(* CoDeSys 2.3.9.42 project: CR0403 AGV.pro *)
(* Libraries: SysLibPlcCtrl.lib 13.6.03 15:49:00, SysLibFile.lib 23.9.04 10:11:36, SysLibTime.lib 27.4.05 10:36:52, SysLibTargetVisu.lib 5.4.04 13:31:00, LinuxSystemLib.Lib 18.3.03 13:26:50, ifm_pdm_file_V010006.lib 14.1.08 14:21:32, ifm_CR0403\ifm_CR0403_V030100.lib 22.3.17 12:39:40, Util.lib 6.11.07 16:39:24, ifm_J1939_NT\ifm_J1939_NT_V020004.lib 18.9.14 16:13:02, ifm_RAWCan\ifm_RAWCan_NT_V020004.lib 3.11.15 19:07:52, standard.lib 4.10.05 11:14:46, SysLibCallback.lib 26.9.08 17:43:52 *)

(* PLC configuration (modules and I/O channels)
Configuration [LocalConfiguration] node 0, in %IB0 out %QB0 {IFM_PARAM_WORD_TIME = 0}
Input/Output [LocalInputOutput] node 1, in %IB0 out %QB0
  Inputs Binary [LocalIn] node 0, in %IB0 out %QB0
    IN00 AT %IB0 [ChInputBool] Input 00 Bit
    IN01 AT %IB1 [ChInputBool] Input 01 Bit
    IN02 AT %IB2 [ChInputBool] Input 02 Bit
    IN03 AT %IB3 [ChInputBool] Input 03 Bit
    IN04 AT %IB4 [ChInputBool] Input 04 Bit
    IN05 AT %IB5 [ChInputBool] Input 05 Bit
    IN06 AT %IB6 [ChInputBool] Input 06 Bit
    IN07 AT %IB7 [ChInputBool] Input 07 Bit
    IN08 AT %IB8 [ChInputBool] Input 08 Bit
    IN09 AT %IB9 [ChInputBool] Input 09 Bit
    IN10 AT %IB10 [ChInputBool] Input 10 Bit
    IN11 AT %IB11 [ChInputBool] Input 11 Bit
  Outputs Binary [LocalOut] node 1, in %IB12 out %QB0
    OUT00 AT %QB0 [ChOutputBool] Output 00 Bit
    OUT01 AT %QB1 [ChOutputBool] Output 01 Bit
    OUT02 AT %QB2 [ChOutputBool] Output 02 Bit
    OUT03 AT %QB3 [ChOutputBool] Output 03 Bit
    OUT04 AT %QB4 [ChOutputBool] Output 04 Bit
    OUT05 AT %QB5 [ChOutputBool] Output 05 Bit
    OUT06 AT %QB6 [ChOutputBool] Output 06 Bit
    OUT07 AT %QB7 [ChOutputBool] Output 07 Bit
    OUT08 AT %QB8 [ChOutputBool] Output 08 Bit
    OUT09 AT %QB9 [ChOutputBool] Output 09 Bit
    OUT10 AT %QB10 [ChOutputBool] Output 10 Bit
    OUT11 AT %QB11 [ChOutputBool] Output 11 Bit
  System Inputs [LocalSystemInputs] node 2, in %IB12 out %QB12
    SUPPLY_VOLTAGE_VBBS AT %IW6 [ChInputWord] Supply voltage VBBS
    SUPPLY_VOLTAGE_VU AT %IW7 [ChInputWord] Supply voltage VU
    SUPPLY_VOLTAGE_VBB1 AT %IW8 [ChInputWord] Supply voltage VBB1
    SUPPLY_VOLTAGE_VBB2 AT %IW9 [ChInputWord] Supply voltage VBB2
    TEMPERATURE AT %IW10 [ChInputInt] Temperature
J1939 Interface [CAN_J1939] node 1, in %IB32 out %QB12
CANopen Interface [CAN_OPEN] node 0, in %IB32 out %QB12
J1939 Interface [CAN_J1939] node 1, in %IB32 out %QB12
*)

(* Global variable list: Global_Variables *)
VAR_GLOBAL
	Route1: ARRAY [1..2,1..4] OF REAL := 10, 100, 100, 10, 10, 10, 100, 100;
END_VAR

(* Data type *)
TYPE CONSTANTS_MATH :
STRUCT
	RadDeg : REAL := 57.29577951; (*Conversie van radialen naar degrees*)
	PI : REAL := 	3.14159265358979323846264338327950288;		(* Kreiszahl PI *)
	PI2 : REAL := 	6.28318530717958647692528676655900576;	(* PI * 2 *)
	PI4 : REAL :=  12.56637061435917295385057353311801152;	(* PI * 4 *)
	PI05 : REAL :=  1.5707963267949;							(* PI / 2 *)
	PI025 : REAL := 0.785398163397448;							(* PI / 4 *)
	PI_INV : REAL := 0.318309886183791;						(* 1 / PI *)
	E : REAL := 	2.71828182845904523536028747135266249;		(* Euler constant e *)
	E_INV : REAL := 0.367879441171442;							(* 1 / e *)
	SQ2 : REAL :=	1.4142135623731;							(* Wurzel von 2 *)
	FACTS : ARRAY[0..12] OF DINT := 1,1,2,6,24,120,720,5040,40320,362880,3628800,39916800,479001600;
END_STRUCT
END_TYPE

(* POU PLC_PRG, ST *)
PROGRAM PLC_PRG
VAR
	CAN_ENABLE_CAN2: CAN_ENABLE;
	CAN_ENABLE_CAN1: CAN_ENABLE;

END_VAR
CAN_ENABLE_CAN1(ENABLE:=TRUE , CHANNEL:=1 , BAUDRATE:=500 , RESULT=> );

CAN_RX_comm_display();

NavSof();

PosEncoderLinks;


PosEncoderRechts;
END_PROGRAM

(* POU CAN_RX_comm_display, ST *)
PROGRAM CAN_RX_comm_display
VAR
	CAN_RX_comm_keys_display: CAN_RX;
	UNPACK_comm_keys: UNPACK;
	keyF1: BOOL;
	keyF2: BOOL;
	keyF3: BOOL;
	keyF4: BOOL;
END_VAR
CAN_RX_comm_keys_display(
	ENABLE:=TRUE ,
	CHANNEL:=1 ,
	ID:=16#190 ,
	DATA=> ,
	RESULT=> );

IF CAN_RX_comm_keys_display.RESULT=1  THEN

UNPACK_comm_keys(
	B:=CAN_RX_comm_keys_display.DATA[0] ,
	B0=>keyF1 ,
	B1=>keyF2 ,
	B2=>keyF3,
	B3=>keyF4 ,
	B4=> ,
	B5=> , 
	B6=> , 
	B7=> );


END_IF

IF keyF1 THEN
OUT00:=TRUE;
ELSE
OUT00:=FALSE;
END_IF

IF keyF2 THEN
OUT01:=TRUE;
ELSE
OUT01:=FALSE;
END_IF
END_PROGRAM

(* POU NavSof, ST *)
PROGRAM NavSof
VAR
	(*Variabelen voor het binnen lezen van de UWB data via de CAN bus*)
	CAN_RX_POZXY_COORD: CAN_RX;							(*FB om een CAN bericht binnen te lezen*)
	ARRAY_TO_DWORD_Xcoor: ARRAY_TO_DWORD;				(*Data van een ARRAY naar een getal omvormen*)
	xHuidigeCoordinaat: REAL;										(*Datatype vastleggen*)
	ARRAY_TO_DWORD_Ycoor: ARRAY_TO_DWORD;
	yHuidigeCoordinaat: REAL;

	(*Variabelen NavSof*)
	i_Waypoints: INT := 0;													(*Variabele die het aantal waypoints van onze huidige route bevat*)
	x_Jumplock: BOOL := TRUE;											(*Flag zodat bij opstart éénmalig X en Y-huidig kunnen gebruikt worden als X en Y start voor de trackline*)
	xStartCoordinaat: REAL := 0;											(*X coordinaat voor begin trackline*)
	yStartCoordinaat: REAL := 0;											(*Y coordinaat voor einde trackline*)
	xEindCoordinaat: REAL := 0;											(*X coordinaat voor einde trackline*)
	yEindCoordinaat: REAL := 0;											(*Y coordinaat voor einde trackline*)
	rAfstandTotWaypoint: REAL := 0;										(*Bevat de afstand tot het waypoint*)
	rTrackHoek: REAL:= 0;												(*Bevat de trackhoek, de hoek die de AGV naar links of rechts doet sturen opdat deze terug op de trackline zou uitkomen*)
	CONSTANTS_MATH: CONSTANTS_MATH;							(*Struct die bepaalde wiskundige constanten bevat*)


	rHoekAGV: REAL;
	rTrack: REAL;
	BNO_lock: BOOL;
	StuurLinks: REAL;
	beginBNO: REAL;
	eindeBNO: REAL;
	StuurNeutraal: REAL;
END_VAR
(*Binnenlezen van de huidige positie d.m.v. UWB*)
CAN_RX_POZXY_COORD(
	ENABLE:= TRUE,
	CHANNEL:=1 ,
	ID:=16#A1 ,
	DATA=> , 
	RESULT=> );

IF  CAN_RX_POZXY_COORD.RESULT=1 THEN

ARRAY_TO_DWORD_Xcoor(
	Byte_0:=CAN_RX_POZXY_COORD.DATA[0] ,
	Byte_1:=CAN_RX_POZXY_COORD.DATA[1] ,
	Byte_2:=CAN_RX_POZXY_COORD.DATA[2] ,
	Byte_3:=CAN_RX_POZXY_COORD.DATA[3] ,
	DWORD_OUT=> xHuidigeCoordinaat );

ARRAY_TO_DWORD_Ycoor(
	Byte_0:=CAN_RX_POZXY_COORD.DATA[4] ,
	Byte_1:=CAN_RX_POZXY_COORD.DATA[5] ,
	Byte_2:=CAN_RX_POZXY_COORD.DATA[6] ,
	Byte_3:=CAN_RX_POZXY_COORD.DATA[7] ,
	DWORD_OUT=> yHuidigeCoordinaat );

END_IF

(*Het aantal waypoints van onze huidige route bepalen*)
i_Waypoints := SIZEOF(Route1)/8;							(*Route 1 bevat 2 * 4 coordinaten die telkens 4 bytes (datatype REAL) innemen
																de totale grootte van deze array is dus 32 bytes / 8 geeft ons het aantal waypoints*)

(*Ervoor zorgen dat bij opstart éénmalig X- en Y-huidig gebruikt kunnen worden als X- en Y-start voor de trackline*)
IF x_Jumplock = TRUE
THEN
	xStartCoordinaat := xHuidigeCoordinaat;
	yStartCoordinaat := yHuidigeCoordinaat;
	x_Jumplock := FALSE;
END_IF;

(*Uitrekenen wat de afstand tot het volgende waypoint is*)
rAfstandTotWaypoint := Afstand_Punt_Punt(xStartCoordinaat, yStartCoordinaat, xEindCoordinaat, yEindCoordinaat);

(*Ervoor zorgen dat bij het afleggen van een route er steeds geweten is of je links of rechts van je trackline zit*)
	rTrack := ATAN2(yStartCoordinaat - yEindCoordinaat , xStartCoordinaat -  xEindCoordinaat )*57.29577951;
	rHoekAGV := ATAN2(yHuidigeCoordinaat - yEindCoordinaat , xHuidigeCoordinaat - xEindCoordinaat )*57.29577951;

IF rTrack < rHoekAGV														(*Onder deze voorwaarde zitten we rechts van onze trackline en moeten we dus naar links sturen*)
THEN
	beginBNO:=0;															(*Hierin moet de waarde van de BNO055 opgeslaan worden*)
	WHILE BNO_lock
	DO
	StuurLinks;															(*Rechtermotor moet meer aangestuurd worden bij tankbesturing of er moet naar links gestuurd worden bij een Ackermansturing*)
		IF ABS(rTrack-rHoekAGV) <= ABS(beginBNO-eindeBNO)		(*Bepaalt hoelang er naar rechts of links moet gestuurd worden*)
		THEN
		BNO_lock := FALSE;												(*Hierdoor wordt het commando om naar links te sturen onderbroken als de gewenste hoek bereikt is*)
		StuurNeutraal;
		END_IF;
	END_WHILE;
END_IF;




Route1[1,1];






(*
rTrackHoek := (ATAN2(yCoor2 - yCoor1,xCoor2 - xCoor1)* CONSTANTS_MATH.RadDeg);
(*ATAN2(Y, X)*)
*)
END_PROGRAM

(* POU FunctiesNavSof/Afstand_Punt_Punt, ST *)
FUNCTION Afstand_Punt_Punt : REAL
VAR_INPUT
	X1 : REAL;
	Y1 : REAL;
	X2 : REAL;
	Y2 : REAL;
END_VAR
VAR
END_VAR
(*****
Doel: Deze functie heeft als doel de afstand tussen twee punten te berekenen
Parameters:
real x1			real y1			real x2			real y2
Return value:
real
*****)

Afstand_Punt_Punt := SQRT(((X2-X1)*(X2-X1))+((Y2-Y1)*(Y2-Y1)));
END_FUNCTION

(* POU FunctiesNavSof/ATAN2, ST *)
FUNCTION ATAN2 : REAL
VAR_INPUT
	Y : REAL;
	X : REAL;
END_VAR
VAR
	MATH: CONSTANTS_MATH;
END_VAR
IF X > 0.0 THEN
	ATAN2 := ATAN(Y/X);
ELSIF X < 0.0 THEN
	IF Y >=0.0 THEN
		ATAN2 := ATAN(Y/X) + MATH.PI;
	ELSE
		ATAN2 := ATAN(Y/X) - MATH.PI;
	END_IF;
ELSIF Y > 0.0 THEN
	ATAN2 := MATH.PI05;
ELSIF Y < 0.0 THEN
	ATAN2 := -MATH.PI05;
ELSE
	ATAN2 := 0.0;
END_IF;


(* revision history hm	20.  apr. 2008	rev 1.0 original version
hm	18. oct. 2008	rev 1.1 	changed to use math constants
hm	10. mar. 2009	rev 1.2	real constants updated to new systax using dot
*)
END_FUNCTION

(* POU FunctiesNavSof/Rico, ST *)
FUNCTION Rico : REAL
VAR_INPUT
	X1 : REAL;
	Y1 : REAL;
	X2 : REAL;
	Y2 : REAL;
END_VAR
VAR
END_VAR
(*****
Doel: De rico berekenen van een rechte gevormd door twee punten
Parameters:
real x1			real y1			real x2			real y2
Return value:
real
*****)

Rico := ((Y2-Y1)/(X2-X1));
END_FUNCTION
